// Output from cart control task
// Input to slave arm control task  
TYPE ST_CartStatus :
STRUCT
	m_CartState :ARRAY[1..g_cartJntNum] OF E_CartJointState:=[g_cartJntNum(CartJointState_Error)];
	
	m_asepticDeployCompletedFlag : BOOL;
	m_inMotion : BOOL := false;
END_STRUCT
END_TYPE

(* stored: Version 1.1.0.1, ProductVersion 3.1.4024.11
   DUT ST_CartStatus: Id {c5c522d4-cd8d-4693-8ddf-cc40ab1df9b3} *)
